(* PLC project Tc2_Standard.CTD Demo, tc3-libraries-kb TwinCAT 3.1 *)
(* stored: creationDateTime 2026-05-10T08:00:00, modificationDateTime 2026-05-10T08:00:00 *)

PROGRAM P_Demo_CTD
  VAR
    fbCTD : CTD;  (* Counter 实例 *)
    bLoad : BOOL;  (* 脉冲一次：把 CV 装入 5 *)
    bCountDown : BOOL;  (* 每给一次上升沿 CV 减 1 *)
    bDone : BOOL;  (* CV 减到 0 时 TRUE *)
    nCV : WORD;  (* 当前剩余计数（监视） *)
  END_VAR

            // ============================================================
// Tc2_Standard.CTD 演示程序
// ============================================================
// 场景：倒计时 5 个产品后置位完成位
// 验证步骤：
//   1. 把本 PROGRAM 加到 PlcTask 调用列表
//   2. 编译并登录目标
//   1. 强制 bLoad := TRUE 一个周期 → nCV 变成 5
//   2. 重复给 bCountDown FALSE → TRUE → FALSE 五次 → nCV 减到 0
//   3. nCV = 0 时观察 bDone 为 TRUE
// ============================================================

fbCTD(
    CD   := bCountDown,
    LOAD := bLoad,
    PV   := WORD#5,
    Q    => bDone,
    CV   => nCV
);

          
END_PROGRAM
